// TwinCAT 3 PLC project test
// ProgramVersion: 3.1.4020.5
// libraries:
//   L2Si Vacuum Library, * (SLAC)
//   LCLS General, * (SLAC)
//   PMPS, * (SLAC - LCLS)
//   Tc2_Standard, * (Beckhoff Automation GmbH)
//   Tc2_System, * (Beckhoff Automation GmbH)
//   Tc2_Utilities, * (Beckhoff Automation GmbH)
//   Tc3_Module, * (Beckhoff Automation GmbH)
// project tree:
//   DUTs/ E_STATES.TcTLEO
//   GVLs/ GVL_Devices.TcGVL, GVL_PMPS.TcGVL
//   / PlcTask.TcTTO
//   POUs/ FB_ValveBase.TcPOU, FB_VGC.TcPOU, FB_VGC_FFO.TcPOU, FB_VRC_NO.TcPOU, MAIN.TcPOU, PRG_VLS.TcPOU
// real-time tasks:
//   TASK PlcTask: cycle T#10ms, priority 20, ADS port 350
//   TASK SimTask: cycle T#10ms, priority 1, ADS port 351
//   TASK VacTask: cycle T#10ms, priority 2, ADS port 352
// I/O:
//   DEVICE Device 1 (EtherCAT) (disabled), AmsNetId 172.21.148.60.2.1
//     Term 1 (EK1100) [EK1100 EtherCAT Coupler (2A E-Bus)]
//       Term 2 (EL3174-0002) [EL3174-0002 4Ch. Ana. Input +/-10V, +/-20mA 16 Bit, Isolated Channels]
//       Term 3 (EL3174-0002) [EL3174-0002 4Ch. Ana. Input +/-10V, +/-20mA 16 Bit, Isolated Channels]
//       Term 4 (EL2624) [EL2624 4Ch. Relay Output, NO (125V AC / 30V DC)]
//       Term 6 (EL1004) [EL1004 4Ch. Dig. Input 24V, 3ms]
//       Term 5 (EL1004) [EL1004 4Ch. Dig. Input 24V, 3ms]
//       Term 7 (EL2004) [EL2004 4Ch. Dig. Output 24V, 0.5A]
//       Term 8 (EL3064) [EL3064 4Ch. Ana. Input 0-10V]
//       Term 9 (EL2794) [EL2794 4Ch. Dig. Output 24V AC/DC, 2A, short-circuit-proof]
//       Term 10 (EL1004) [EL1004 4Ch. Dig. Input 24V, 3ms]
//       Term 11 (EL1124) [EL1124 4Ch. Dig. Input 5V, 10µs, Sensor Power]
//       Term 12 (EL1124) [EL1124 4Ch. Dig. Input 5V, 10µs, Sensor Power]
//       Term 13 (EL3064) [EL3064 4Ch. Ana. Input 0-10V]
// variable links:
//   SIM/SIM Instance <-> test/test Instance
//     PlcTaskSim Inputs/GVL_SimDevices.S_FEE_GCC_03.i_xHvOn <-> PlcTask Outputs/GVL_Devices.FEE_GCC_03.q_xHV_DIS
//     PlcTaskSim Inputs/GVL_SimDevices.S_FEE_GCC_04.i_xHvOn <-> PlcTask Outputs/GVL_Devices.FEE_GCC_04.q_xHV_DIS
//     PlcTaskSim Inputs/GVL_SimDevices.S_FEE_KMONO_GCC_01.i_xHvOn <-> PlcTask Outputs/GVL_Devices.FEE_KMONO_GCC_01.q_xHV_DIS
//     PlcTaskSim Inputs/GVL_SimDevices.S_FEE_KMONO_PIP_01.xOn <-> PlcTask Outputs/GVL_Devices.FEE_KMONO_PIP_01.q_xHVEna_DO
//     PlcTaskSim Inputs/GVL_SimDevices.S_FEE_M1L_PIP_01.xOn <-> PlcTask Outputs/GVL_Devices.FEE_M1L_PIP_01.q_xHVEna_DO
//     PlcTaskSim Inputs/GVL_SimDevices.S_FEE_MIL_GCC_02.i_xHvOn <-> PlcTask Outputs/GVL_Devices.FEE_M1L_GCC_01.q_xHV_DIS
//     PlcTaskSim Inputs/GVL_SimDevices.S_FEE_PIP_02.xOn <-> PlcTask Outputs/GVL_Devices.FEE_PIP_02.q_xHVEna_DO
//     PlcTaskSim Inputs/GVL_SimDevices.S_FEE_PIP_03.xOn <-> PlcTask Outputs/GVL_Devices.FEE_PIP_03.q_xHVEna_DO
//     PlcTaskSim Inputs/GVL_SimDevices.S_FEE_VGC_02.i_xSol <-> PlcTask Outputs/GVL_Devices.FEE_VGC_02.q_xOPN_DO
//     PlcTaskSim Inputs/GVL_SimDevices.S_FEE_VGC_03.i_xSol <-> PlcTask Outputs/GVL_Devices.FEE_VGC_03.q_xOPN_DO
//     PlcTaskSim Inputs/GVL_SimDevices.S_FEE_VGC_04.i_xSol <-> PlcTask Outputs/GVL_Devices.FEE_VGC_04.q_xOPN_DO
//     PlcTaskSim Inputs/GVL_SimDevices.VGC_1.i_xSol <-> PlcTask Outputs/PRG_VLS.VGC_1.q_xOPN_DO
//     PlcTaskSim Inputs/GVL_SimDevices.VGC_W.i_xSol <-> PlcTask Outputs/PRG_VLS.VGC_W.q_xCLS_DO
//     PlcTaskSim Outputs/GVL_SimDevices.S_FEE_GCC_03.q_DisActive <-> PlcTask Inputs/GVL_Devices.FEE_GCC_03.i_xDisc_Active
//     PlcTaskSim Outputs/GVL_SimDevices.S_FEE_GCC_04.q_DisActive <-> PlcTask Inputs/GVL_Devices.FEE_GCC_04.i_xDisc_Active
//     PlcTaskSim Outputs/GVL_SimDevices.S_FEE_GCC_03.q_iRawPress <-> PlcTask Inputs/GVL_Devices.FEE_GCC_03.i_iPRESS_R
//     PlcTaskSim Outputs/GVL_SimDevices.S_FEE_GCC_04.q_iRawPress <-> PlcTask Inputs/GVL_Devices.FEE_GCC_04.i_iPRESS_R
//     PlcTaskSim Outputs/GVL_SimDevices.S_FEE_GCC_03.q_iRawPress <-> PlcTask Inputs/PRG_VLS.DS_GCC.i_iPRESS_R
//     PlcTaskSim Outputs/GVL_SimDevices.S_FEE_GCC_03.q_xHVOn <-> PlcTask Inputs/GVL_Devices.FEE_GCC_03.i_xHV_ON
//     PlcTaskSim Outputs/GVL_SimDevices.S_FEE_GCC_04.q_xHVOn <-> PlcTask Inputs/GVL_Devices.FEE_GCC_04.i_xHV_ON
//     PlcTaskSim Outputs/GVL_SimDevices.S_FEE_GPI_03.q_iRawPress <-> PlcTask Inputs/GVL_Devices.FEE_GPI_03.i_iPRESS_R
//     PlcTaskSim Outputs/GVL_SimDevices.S_FEE_GPI_04.q_iRawPress <-> PlcTask Inputs/GVL_Devices.FEE_GPI_04.i_iPRESS_R
//     PlcTaskSim Outputs/GVL_SimDevices.S_FEE_GPI_03.q_iRawPress <-> PlcTask Inputs/PRG_VLS.DS_GPI.i_iPRESS_R
//     PlcTaskSim Outputs/GVL_SimDevices.S_FEE_KMONO_GCC_01.q_DisActive <-> PlcTask Inputs/GVL_Devices.FEE_KMONO_GCC_01.i_xDisc_Active
//     PlcTaskSim Outputs/GVL_SimDevices.S_FEE_KMONO_GCC_01.q_iRawPress <-> PlcTask Inputs/GVL_Devices.FEE_KMONO_GCC_01.i_iPRESS_R
//     PlcTaskSim Outputs/GVL_SimDevices.S_FEE_KMONO_GCC_01.q_iRawPress <-> PlcTask Inputs/PRG_VLS.US_GCC.i_iPRESS_R
//     PlcTaskSim Outputs/GVL_SimDevices.S_FEE_KMONO_GCC_01.q_xHVOn <-> PlcTask Inputs/GVL_Devices.FEE_KMONO_GCC_01.i_xHV_ON
//     PlcTaskSim Outputs/GVL_SimDevices.S_FEE_KMONO_GPI_01.q_iRawPress <-> PlcTask Inputs/GVL_Devices.FEE_KMONO_GPI_01.i_iPRESS_R
//     PlcTaskSim Outputs/GVL_SimDevices.S_FEE_KMONO_GPI_01.q_iRawPress <-> PlcTask Inputs/PRG_VLS.US_GPI.i_iPRESS_R
//     PlcTaskSim Outputs/GVL_SimDevices.S_FEE_M1L_GPI_02.q_iRawPress <-> PlcTask Inputs/GVL_Devices.FEE_M1L_GPI_01.i_iPRESS_R
//     PlcTaskSim Outputs/GVL_SimDevices.S_FEE_MIL_GCC_02.q_DisActive <-> PlcTask Inputs/GVL_Devices.FEE_M1L_GCC_01.i_xDisc_Active
//     PlcTaskSim Outputs/GVL_SimDevices.S_FEE_MIL_GCC_02.q_iRawPress <-> PlcTask Inputs/GVL_Devices.FEE_M1L_GCC_01.i_iPRESS_R
//     PlcTaskSim Outputs/GVL_SimDevices.S_FEE_MIL_GCC_02.q_xHVOn <-> PlcTask Inputs/GVL_Devices.FEE_M1L_GCC_01.i_xHV_ON
//     PlcTaskSim Outputs/GVL_SimDevices.S_FEE_VGC_02.q_xClsLS <-> PlcTask Inputs/GVL_Devices.FEE_VGC_02.i_xClsLS
//     PlcTaskSim Outputs/GVL_SimDevices.S_FEE_VGC_03.q_xClsLS <-> PlcTask Inputs/GVL_Devices.FEE_VGC_03.i_xClsLS
//     PlcTaskSim Outputs/GVL_SimDevices.S_FEE_VGC_04.q_xClsLS <-> PlcTask Inputs/GVL_Devices.FEE_VGC_04.i_xClsLS
//     PlcTaskSim Outputs/GVL_SimDevices.S_FEE_VGC_02.q_xOpnLS <-> PlcTask Inputs/GVL_Devices.FEE_VGC_02.i_xOpnLS
//     PlcTaskSim Outputs/GVL_SimDevices.S_FEE_VGC_03.q_xOpnLS <-> PlcTask Inputs/GVL_Devices.FEE_VGC_03.i_xOpnLS
//     PlcTaskSim Outputs/GVL_SimDevices.S_FEE_VGC_04.q_xOpnLS <-> PlcTask Inputs/GVL_Devices.FEE_VGC_04.i_xOpnLS
//     PlcTaskSim Outputs/GVL_SimDevices.VGC_1.q_xClsLS <-> PlcTask Inputs/PRG_VLS.VGC_1.i_xClsLS
//     PlcTaskSim Outputs/GVL_SimDevices.VGC_1.q_xOpnLS <-> PlcTask Inputs/PRG_VLS.VGC_1.i_xOpnLS
//     PlcTaskSim Outputs/GVL_SimDevices.VGC_W.q_xClsLS <-> PlcTask Inputs/PRG_VLS.VGC_W.i_xClsLS
//     PlcTaskSim Outputs/GVL_SimDevices.VGC_W.q_xOpnLS <-> PlcTask Inputs/PRG_VLS.VGC_W.i_xOpnLS

CONFIGURATION test
    RESOURCE PLC ON TwinCAT3
        TASK PlcTask(INTERVAL := T#10ms, PRIORITY := 2);
        PROGRAM MAIN WITH PlcTask : MAIN;
    END_RESOURCE
END_CONFIGURATION

// ---- DUTs/E_STATES.TcTLEO
{attribute 'qualified_only'}
{attribute 'strict'}
TYPE E_STATES :
(
	INIT := 0, // INIT 
	NOT_SAFE ,// NOT OK to move in the same state
	READY, // Safe to Move STATE
	OVERRIDE,
	SETUP
	
);
END_TYPE

// ---- GVLs/GVL_Devices.TcGVL
VAR_GLOBAL
	
	

/////////////////////
	{attribute 'pytmc' := '
    pv: FEE:VGC:02
	'}
	FEE_VGC_02: FB_VGC;
	{attribute 'pytmc' := '
    pv: FEE:KMONO:GPI:01
	'}
	FEE_KMONO_GPI_01: FB_MKS275;
	{attribute 'pytmc' := '
    pv: FEE:KMONO:GCC:01
	'}
	FEE_KMONO_GCC_01: FB_MKS500;
	{attribute 'pytmc' := '
    pv: FEE:KMONO:PIP:01
	'}
	FEE_KMONO_PIP_01: FB_PIP_Gamma;
	{attribute 'pytmc' := '
    pv: FEE:PIP:02
	'}
	FEE_PIP_02: FB_PIP_Gamma;
	{attribute 'pytmc' := '
    pv: FEE:GPI:03
	'}
	FEE_GPI_03: FB_MKS275;
	{attribute 'pytmc' := '
    pv: FEE:GCC:03
	'}
	FEE_GCC_03: FB_MKS500;
	{attribute 'pytmc' := '
    pv: FEE:VGC:03
	'}
	FEE_VGC_03: FB_VGC_FFO;
	{attribute 'pytmc' := '
    pv: FEE:M1L:GPI:01
	'}
	FEE_M1L_GPI_01: FB_MKS275;
	{attribute 'pytmc' := '
    pv: FEE:M1L:GCC:03
	'}
	FEE_M1L_GCC_01: FB_MKS500;
	{attribute 'pytmc' := '
    pv: FEE:M1L:PIP:01
	'}
	FEE_M1L_PIP_01: FB_PIP_Gamma;
	{attribute 'pytmc' := '
    pv: FEE:PIP:03
	'}
	FEE_PIP_03: FB_PIP_Gamma;
	{attribute 'pytmc' := '
    pv: FEE:GPI:04
	'}
	FEE_GPI_04: FB_MKS275;
	{attribute 'pytmc' := '
    pv: FEE:GCC:04
	'}
	FEE_GCC_04: FB_MKS500;
	{attribute 'pytmc' := '
    pv: FEE:VGC:04
	'}
	FEE_VGC_04: FB_VGC_FFO;
	
END_VAR

// ---- GVLs/GVL_PMPS.TcGVL

VAR_GLOBAL
	
{attribute 'pytmc' := '
    pv: PLC:TST:FF1
    '}
    {attribute 'TcLinkTo' := '.q_xFastFaultOut:=TIIB[PMPS_FFO]^Channel 1^Output'}
    g_FastFaultOutput1  :   FB_HardwareFFOutput;
	
	{attribute 'pytmc' := '
    pv: PLC:TST:FF2
    '}
    {attribute 'TcLinkTo' := '.q_xFastFaultOut:=TIIB[PMPS_FFO]^Channel 2^Output'}
    g_FastFaultOutput2  :   FB_HardwareFFOutput;
END_VAR

// ---- POUs/MAIN.TcPOU
PROGRAM MAIN
VAR
	
	

END_VAR

PRG_VLS();

//valves
FEE_VGC_02(
	i_stUSG:= FEE_KMONO_GCC_01.IG, 
	i_stDSG:= FEE_KMONO_GCC_01.IG , 
	i_xDis_DPIlk:= FALSE, 
	i_xEPS_OPN_OK:= , 
	i_xEPS_CLS_OK:= ,
	i_xPMPS_OK:= , 
	i_xExt_OK:= TRUE, 
	i_xOverrideMode:= , 
	i_xReset:= , 
	iq_stValve=>);

FEE_VGC_03(
	i_stUSG:=FEE_KMONO_GCC_01.IG, 
	i_stDSG:= FEE_M1L_GCC_01.IG , 
	i_xDis_DPIlk:= FALSE, 
	i_xEPS_OPN_OK:= TRUE, 
	i_xEPS_CLS_OK:= TRUE,
	i_xPMPS_OK:= TRUE, 
	i_xExt_OK:= TRUE, 
	i_xOverrideMode:= , 
	i_xReset:= , 
	iq_stValve=> , 
	xMPS_OK=> , 
	io_fbFFHWO:= g_FastFaultOutput1 );

FEE_VGC_04(
	i_stUSG:= FEE_GCC_03.IG, 
	i_stDSG:= FEE_GCC_03.IG , 
	i_xDis_DPIlk:= FALSE, 
	i_xEPS_OPN_OK:= TRUE, 
	i_xEPS_CLS_OK:= TRUE,
	i_xPMPS_OK:= TRUE, 
	i_xExt_OK:= TRUE, 
	i_xOverrideMode:= , 
	i_xReset:= , 
	iq_stValve=> , 
	xMPS_OK=> , 
	io_fbFFHWO:= g_FastFaultOutput2 );	
	
// gauges and pip
FEE_KMONO_GPI_01(PG=>);
FEE_KMONO_GCC_01(PG:=FEE_KMONO_GPI_01.PG);
FEE_KMONO_PIP_01(i_stGauge:= FEE_KMONO_GCC_01.IG);

FEE_GPI_03(PG=>);
FEE_GCC_03(PG:=FEE_KMONO_GPI_01.PG);

FEE_PIP_02(i_stGauge:= FEE_GCC_03.IG);

FEE_M1L_GPI_01(PG=>);
FEE_M1L_GCC_01(PG:=FEE_M1L_GPI_01.PG);
FEE_M1L_PIP_01(i_stGauge:= FEE_M1L_GCC_01.IG);

FEE_GPI_04(PG=>);
FEE_GCC_04(PG:=FEE_GPI_04.PG);
FEE_PIP_03(i_stGauge:= FEE_GCC_04.IG);



/// fast fault

g_FastFaultOutput1.EvaluateOutput(i_xVeto:=PMPS_GVL.stCurrentBeamParameters.aStoppers[PMPS.L_Stopper.ST1]);
g_FastFaultOutput2.EvaluateOutput(i_xVeto:=PMPS_GVL.stCurrentBeamParameters.aStoppers[PMPS.L_Stopper.ST1]);

END_PROGRAM

// ---- POUs/PRG_VLS.TcPOU
PROGRAM PRG_VLS
VAR
	xFirstPass	:	BOOL;
	fbFSInit		:	R_TRIG;
	
	state:E_STATES;
	

	bOverride:BOOL;
	bSetup:BOOL;
	
	
	//GVL_Devices
	VGC_1	:FB_VGC;
	VGC_W	:FB_VRC_NO; // Is the Window valve NO 

	US_GPI: FB_MKS275;
	US_GCC: FB_MKS422;

	DS_GPI: FB_MKS275;
	DS_GCC: FB_MKS422;
END_VAR

fbFSInit( CLK := TRUE, Q => xFirstPass);
(* On first PLC pass, put valve into init state*)
IF xFirstPass THEN
	state:= E_STATES.INIT;
	bOverride := FALSE;
	bSetup := FALSE;
END_IF


//STATE ACTIONS
CASE state OF

 E_STATES.INIT: 
		VGC_1.M_Set_OPN_SW(FALSE); //Isolation Valve closed
		VGC_W.M_Set_CLS_SW(FALSE); // Window valve OPEN
		VGC_1.i_xOverrideMode := VGC_W.i_xOverrideMode := FALSE;
		//Transition
		if (VGC_1.M_IsClosed() AND VGC_W.M_IsOpen()) THEN
			state:= E_STATES.NOT_SAFE;
		END_IF
		
E_STATES.NOT_SAFE: // System is not allowed to actuate, i.e all interlocks are in effect
 	VGC_1.i_xExt_OK := VGC_1.i_xEPS_OPN_OK := VGC_1.i_xEPS_CLS_OK:= FALSE; 
	VGC_W.i_xExtILK_OK:= FALSE; 
	VGC_1.i_xOverrideMode := VGC_W.i_xOverrideMode := FALSE;

	//Transition
	if (US_GCC.IG.xAT_VAC AND DS_GCC.IG.xAT_VAC) THEN state:= E_STATES.READY; END_IF
	
	
 E_STATES.READY: // OK to MOVE
 	// Release the external interlock so the differential pressure inlk is in effect
 	VGC_1.i_xExt_OK:= VGC_1.i_xEPS_OPN_OK := VGC_1.i_xEPS_CLS_OK:= TRUE; 
	//permission to insert window valve only when US vacuum is good??
	VGC_W.i_xExtILK_OK:= US_GCC.IG.xPRESS_OK AND  US_GCC.IG.xAT_VAC; // OR should it be a pressure setpoint
	//Insertion of window valve is followed by automatic openeing of isolation valve.
	// Valves  alternate positions.
	If (VGC_W.M_IsClosed()) THEN  VGC_1.M_Set_OPN_SW(TRUE);
	ELSIF (VGC_W.M_IsOpen()) THEN VGC_1.M_Set_OPN_SW(FALSE);
	END_IF
	
 
 E_STATES.OVERRIDE: 
	// Override Mode is enabled for all valves
 	VGC_1.i_xOverrideMode :=VGC_W.i_xOverrideMode := TRUE;
	// Exit of Override mode always goes back to init
 	IF NOT(bOverride) THEN state:= E_STATES.INIT; END_IF
	
	
 E_STATES.SETUP: 
	// Window valve remains retracted
 	VGC_W.i_xExtILK_OK := FALSE; 
	// Isolation valves operates like standard gate valves 
	VGC_1.i_xExt_OK := TRUE;
	// exit to init just to be safe?
	IF NOT(bSetup) THEN state:= E_STATES.INIT; END_IF
END_CASE





// STATE TRANSITIONS
// the system can go to setup state from any other state except override
IF (bSetup) AND (state<>E_STATES.OVERRIDE) THEN state:= E_STATES.SETUP; 
// the system can go to override state from any other state except setup
ELSIF (bOverride) AND (state<>E_STATES.SETUP) THEN state:= E_STATES.OVERRIDE;
//Loss of at vac signal makes the system go to init/not safe to move state
ELSIF (NOT US_GCC.IG.xAT_VAC ) OR (NOT DS_GCC.IG.xAT_VAC) THEN state:= E_STATES.INIT;
END_IF 





// Instantiate function blocks
US_GPI(PG=>);
US_GCC(PG:=US_GPI.PG);
DS_GPI(PG=>);
DS_GCC(PG:=US_GPI.PG);

VGC_1(
	i_stUSG:= US_GCC.IG, 
	i_stDSG:= DS_GCC.IG , 
	i_xDis_DPIlk:= FALSE, 
	i_xEPS_OPN_OK:= , 
	i_xEPS_CLS_OK:= ,
	i_xPMPS_OK:= , 
	i_xExt_OK:= , 
	i_xOverrideMode:= , 
	i_xReset:= , 
	iq_stValve=>);

VGC_W(i_xExtILK_OK:= , 
	i_xOverrideMode:= ,
    iq_stValve=> );

END_PROGRAM

// ---- POUs/FB_VGC.TcPOU
(* This function block implements basic functionality for Isolation Gate Valves*)
(* This function block interlock is as follows:
1. The valve can be opened when the difference between the pressures on both sides is
less than the maximum differential pressure.
2. This rule persists until the pressures on both sides are lower than the vacuum-setpoint.
3. Once at-vac, the valve will close if the pressure on either side rises above the setpoint.*)
(*This function block also implements PMPS and EPS interlocks, as well as Fast MPS trigger*)
FUNCTION_BLOCK FB_VGC Extends FB_ValveBase
VAR_IN_OUT
END_VAR
VAR_INPUT
	(*Upstream Gauge, usually ion gauge*)
	i_stUSG	:	ST_VG;
	(*Downstream Gauge, usually ion gauge*)
	i_stDSG	:	ST_VG;
	{attribute 'pytmc' := '
    pv: Dis_DPIlk
	'}
	i_xDis_DPIlk : BOOL := FALSE;  (* Set to true when calling the function to disable the differential pressure interlock *)
	{attribute 'pytmc' := '
    pv: EPS_OPN_OK
	'}
	i_xEPS_OPN_OK:	BOOL	:= TRUE; (*External EPS interlock, Set to TRUE when no EPS interlock is required, otherwise set to correct interlock signal*)
	{attribute 'pytmc' := '
    pv: EPS_CLS_OK
	'}
	i_xEPS_CLS_OK:	BOOL	:= TRUE; (*External EPS interlock, Set to TRUE when no EPS interlock is required, otherwise set to correct interlock signal*)
	
	{attribute 'pytmc' := '
    pv: MPS_OK
	'}
	i_xPMPS_OK:	BOOL	; (*External MPS interlock, Set to TRUE when no PMPS interlock is required*)
	i_xExt_OK: BOOL; (*Other External Interlock, Set to True when no external interlock is required. If this Valve is neigboring a Fast Shutter this should be linked to the fast shutter xVAC_FAULT_OK*)
	i_xOverrideMode : BOOL; (*To be linked to global override bit. This Overrides Vacuum logic only, EPS, MPS and PMPS are still enforces*)
	// Reset fault
	{attribute 'pytmc' := '
    pv: FF_Reset
	'}
    i_xReset: BOOL;
END_VAR
VAR_OUTPUT
	{attribute 'pytmc' := '
    pv:
	'}
	iq_stValve : ST_VGC; (* All valve data and states will be in this struct*)
	
END_VAR

VAR
	{attribute 'instance-path'}
	{attribute 'noinit'}
	sPath: STRING;
	rDiffPressAllowed	:	REAL := 22.5; // Torr, Default value comes from Vat Valve Manual
	rDiffPress : REAL;
	set : BOOL;
    reset: BOOL;
	  
	xFirstPass	:	BOOL;
	fbFSInit		:	R_TRIG;
	
	tonDelOK : TON;
	rtOK	:	R_TRIG;
	tonOvrd	:	TON;
	rtOpen	:	R_TRIG;
	ftClose: F_TRIG;
	
	tDelOK	:	TIME := T#60S;
	tOvrd	:	TIME := T#10s;
	ePrevState : E_VGC;
	
	(* Timeouts*)
	tTimeOutDuration: TIME:= T#10S;
	tOPNtimeout: TON;
	tCLStimeout:TON;
	
	
	
	(*IO*)
	i_xOpnLS	AT%I*: BOOL;
	i_xClsLS	AT%I*: BOOL;
	q_xOPN_DO	AT%Q*: BOOL;
    
  
END_VAR

(* Vacuum gate valve
A. Wallace
16-10-29

A gate valve isolates vacuum volumes. Ideally it can be opened when a system is vented
to allow for faster pumping, and will close when high vacuum is lost.

The following behavior is good for valves in something like a gas attenuator.
This function block does the following:
1. The valve can be opened when the difference between the pressures on both sides is
less than the maximum differential pressure.
2. This rule persists until the pressures on both sides are lower than the vacuum-setpoint.
3. Once at-vac, the valve will close if the pressure on either side rises above the setpoint.

Alternatively, the differential pressure interlock can be disabled so the valve may only be opened
if the pressure on both sides is lower than the at-vacuum-setpoint. You want this behavior if 
the valve is to be used in a UHV section.

Hysteresis is employed to ensure a smooth transition from vented/pumping down, to at-vac.

Finally, an override system is built in so you can bypass all the interlocking logic and 
get back online.
*)
(* 10/1/2018 Margaret Ghaly included EPS, PMPS Checkes and MPS trigger signals*)

ACT_Init();
(*IO Mapping*)
ACT_IO();
A_Override();
A_PositionCheck();
ACT_ResetAlarms();
A_EPS();
// Main logic the very last call right before IO
ACT_Main();
(*IO Mapping*)
ACT_IO();
A_Logger();

ACTION A_EPS:
ftClose(CLK:= iq_stValve.pv_xOPN_SW);
rtOpen(CLK:= iq_stValve.pv_xOPN_SW);


(* If Epics Command to close the Valve, check if PMPS and EPS are ok, otherwise Keep command set to open valve *)
// Check a falling edge on the open switch, which means that the valve is commanded to close
IF (ftClose.Q) THEN
	// check that the valve is allowed to close, and that it was already in the open position otherwise, he command is to be ingonred and reset
	IF NOT(i_xEPS_CLS_OK) AND (iq_stValve.q_xOPN_DO) THEN iq_stValve.pv_xOPN_SW := TRUE; END_IF;
END_IF

// if switch pv has been switched to open
IF (rtOpen.Q) THEN 
	// if the EPS interlock the valve from openening, the switch pv is reset to false i.e ignoring the action
	IF NOT (i_xEPS_OPN_OK) THEN  iq_stValve.pv_xOPN_SW := FALSE; END_IF
END_IF
END_ACTION

ACTION A_Logger:
// Log valve timeouts
tErrorPresent(CLK:=iq_stValve.bErrorPresent);
IF tErrorPresent.Q THEN fbLogger(sMsg:=iq_stValve.sErrorMessage, eSevr:=TcEventSeverity.Warning); END_IF

// Log valve open
tAction(CLK:= iq_stValve.q_xOPN_DO);
IF tAction.Q THEN fbLogger(sMsg:='Valve commanded open', eSevr:=TcEventSeverity.Info); END_IF

// Log override mode enabled
tOverrideActivated(CLK:= (tonOvrd.Q AND i_xOverrideMode));
IF tOverrideActivated.Q THEN fbLogger(sMsg:='Valve override mode activated', eSevr:=TcEventSeverity.Warning); END_IF
END_ACTION

ACTION A_Override:
(* Override logic *)
(* Goal: give ability to override, but do so in a way that people won't forget it.
Solution: Override only after ten seconds of override, protect against blips,
when the valve permission goes true for more than ten seconds consistently, remove override
*)

tonDelOK(IN:=iq_stValve.xOPN_OK, PT:=tDelOK);
rtOK(CLK:=tonDelOK.Q);
IF rtOK.Q AND iq_stValve.pv_xOvrdOpn THEN 
	if (iq_stValve.eState = OPEN) AND (i_xOverrideMode) AND (iq_stValve.pv_xOvrdOpn) THEN iq_stValve.pv_xOPN_SW := TRUE; END_IF //for seamless transition   
   	iq_stValve.pv_xOvrdOpn :=FALSE; // reset the overrride open bit
	//Log
    fbLogger(sMsg:='Override expired', eSevr:=TcEventSeverity.Warning);
    
END_IF

//Override timer
tonOvrd(IN:=iq_stValve.pv_xOvrdOpn, PT:=tOvrd);
END_ACTION

ACTION A_PositionCheck:


///Check valve position
IF iq_stValve.i_xClsLS AND  iq_stValve.i_xOpnLS THEN
	iq_stValve.eState:=INVALID;
ELSIF NOT iq_stValve.i_xClsLS AND iq_stValve.i_xOpnLS AND iq_stValve.q_xOPN_DO THEN 
	iq_stValve.eState:=OPEN;
ELSIF iq_stValve.i_xClsLS AND NOT iq_stValve.i_xOpnLS AND NOT iq_stValve.q_xOPN_DO THEN 
	iq_stValve.eState:=CLOSED;
ELSIF NOT iq_stValve.i_xClsLS AND NOT iq_stValve.i_xOpnLS THEN 
	iq_stValve.eState:=MOVING;
ELSE
	iq_stValve.eState:=INVALID;
END_IF


///Check valve moving postion timout
IF NOT iq_stValve.i_xClsLS AND tCLStimeout.Q THEN 
	iq_stValve.bErrorPresent := TRUE;
	iq_stValve.sErrorMessage := ' Close Timeout';
ELSIF NOT iq_stValve.i_xOpnLS AND tOPNtimeout.Q THEN 
	iq_stValve.bErrorPresent := TRUE; 
	iq_stValve.sErrorMessage := ' Open Timeout';
END_IF
IF (iq_stValve.eState=INVALID) THEN
	iq_stValve.bErrorPresent := TRUE; 
	iq_stValve.sErrorMessage := CONCAT(sPath,' Invalid Valve Position');
END_IF


(*Timers*)
tOPNtimeout(IN:= iq_stValve.q_xOPN_DO, PT := tTimeOutDuration );
tCLStimeout(IN:= NOT iq_stValve.q_xOPN_DO, PT := tTimeOutDuration);
END_ACTION

ACTION ACT_Init:
fbFSInit( CLK := TRUE, Q => xFirstPass);
(* On first PLC pass, put valve into vented state, which implies a closed valve *)
IF xFirstPass THEN
	iq_stValve.eVGC_State := Vented;
	iq_stValve.pv_xOPN_SW := FALSE;
END_IF
END_ACTION

ACTION ACT_IO:
(*inputs*)
iq_stValve.i_xOpnLS := 	i_xOpnLS;
iq_stValve.i_xClsLS:=	i_xClsLS;
iq_stValve.xEXT_OK := i_xEXT_OK;
iq_stValve.xOverrideMode := i_xOverrideMode;
(*outputs*)
q_xOPN_DO:= iq_stValve.q_xOPN_DO;
END_ACTION

ACTION ACT_Main:

// Update hysteresis
///////////////////////////////////////////////////
IF iq_stValve.rAT_VAC_SP_LAST <> iq_stValve.rAT_VAC_SP OR xFirstPass THEN
	iq_stValve.rAT_VAC_SP_LAST := iq_stValve.rAT_VAC_SP;
	iq_stValve.rAT_VAC_HYS := iq_stValve.rHYST_PERC * iq_stValve.rAT_VAC_SP;
END_IF

iq_stValve.rAT_VAC_HYS := LIMIT(0, iq_stValve.rAT_VAC_HYS, iq_stValve.rAT_VAC_SP);
IF iq_stValve.rAT_VAC_SP <> 0 THEN
	IF iq_stValve.rHYST_PERC <> (iq_stValve.rAT_VAC_HYS / iq_stValve.rAT_VAC_SP) THEN
		iq_stValve.rHYST_PERC := LIMIT(0, (iq_stValve.rAT_VAC_HYS / iq_stValve.rAT_VAC_SP) ,1);
	END_IF
END_IF
// Valve at vacuum check
///////////////////////////////////////////////////
	set := i_stUSG.rPRESS < iq_stValve.rAT_VAC_HYS AND i_stDSG.rPRESS < iq_stValve.rAT_VAC_HYS AND i_stUSG.xPRESS_OK AND i_stDSG.xPRESS_OK;
 	iq_stValve.xAT_VAC S= set;
	reset := i_stUSG.rPRESS > iq_stValve.rAT_VAC_SP OR i_stDSG.rPRESS > iq_stValve.rAT_VAC_SP OR NOT i_stUSG.xPRESS_OK OR NOT i_stDSG.xPRESS_OK;
	iq_stValve.xAT_VAC R= reset;
	
// Differential pressure check
///////////////////////////////////////////////////
	(* Calc the differential pressure across the valve *)
	rDiffPress := ABS(i_stUSG.rPRESS - i_stDSG.rPRESS);
	
	(* As long as the differential pressure is less than 30mbar, the valve is allowed to open *)
	IF rDiffPress <= rDiffPressAllowed AND i_stUSG.xPRESS_OK AND i_stDSG.xPRESS_OK THEN
		iq_stValve.xDP_OK := TRUE;
	ELSE
		iq_stValve.xDP_OK	:= FALSE;
		(* If the differential pressure is exceeded, even when the valve is open,
		the state is unexpected and triggers a fault, because it suggests that something
		is wrong with the valve, or gauges or mapping or there is a major leak on one side.*)
		iq_stValve.eVGC_State := ERR_DiffPress;
        iq_stValve.xERR_DifPres := TRUE;
	END_IF

// Valve state
///////////////////////////////////////////////////
CASE iq_stValve.eVGC_State OF
	Vented: (* The Vented state is used during pump down *)
        //Log new state
        IF ePrevState <> iq_stValve.eVGC_State THEN
            fbLogger(sMsg:='Vented', eSevr:=TcEventSeverity.Info);
            ePrevState := iq_stValve.eVGC_State;
		END_IF
        
		(* Assuming the pump down went well, we are now at vacuum on both sides,
		so we move to the vacuum state, otherwise remain in the vented state *)
		IF iq_stValve.xAT_VAC AND (NOT (iq_stValve.xERR_DifPres)) AND NOT (NOT (iq_stValve.xERR_SP)) and NOT (NOT (iq_stValve.xERR_ExtFault))THEN
		    iq_stValve.eVGC_State := AtVacuum;
		ELSE
		    iq_stValve.eVGC_State := Vented;
		END_IF
	
	AtVacuum:
        //Log new state
        IF ePrevState <> iq_stValve.eVGC_State THEN
            fbLogger(sMsg:='Vacuum setpoint satisfied', eSevr:=TcEventSeverity.Info);
            ePrevState := iq_stValve.eVGC_State;
		END_IF
        
		IF iq_stValve.xAT_VAC THEN
		(* If both pressure setpoints are made,
		then enable the differential pressure interlock, regardless of the valve state
		assuming we're using some kind of ion gauge where a pressure setpoint cannot be higher than 1E-4 T *)
		iq_stValve.eVGC_State := AtVacuum;
				
		ELSE
		
			(* If the valve is open (or in an unknown state) and either gauge is not at it's vacuum setpoint,
			we have a loss of vacuum error *)
			IF (iq_stValve.i_xOpnLS OR (NOT iq_stValve.i_xOpnLS AND NOT iq_stValve.i_xClsLS)) THEN
				iq_stValve.eVGC_State := ERR_LostVac;
				iq_stValve.xERR_SP := TRUE; //TAW changed this to the ERR_SP bool because I think that's what it was intended to be?
		
			(* Alternatively, if the valve is already closed and we lose pressure on one side,
			it was probably intentional venting, so we calmly move back to venting mode, and
			disable the differential pressure interlock *) //?? 
			ELSIF iq_stValve.i_xClsLS THEN
				iq_stValve.eVGC_State := Vented;
			END_IF
		
		END_IF
	
	ERR_DiffPress:
        //Log new state
        IF ePrevState <> iq_stValve.eVGC_State THEN
            fbLogger(sMsg:='Potential accidental vent.', eSevr:=TcEventSeverity.Critical);
            ePrevState := iq_stValve.eVGC_State;
		END_IF
        
		IF NOT (iq_stValve.xERR_DifPres) THEN
			iq_stValve.eVGC_State := Vented;
		END_IF
		
	
	ERR_LostVac:
        //Log new state
        IF ePrevState <> iq_stValve.eVGC_State THEN
            fbLogger(sMsg:='Unexpected loss of vacuum while valve was open.', eSevr:=TcEventSeverity.Critical);
            ePrevState := iq_stValve.eVGC_State;
		END_IF
		IF NOT (iq_stValve.xERR_SP) THEN
			iq_stValve.eVGC_State := Vented;
		END_IF
		
	ERR_ExtFault:
        //Log new state
        IF ePrevState <> iq_stValve.eVGC_State THEN
            fbLogger(sMsg:='Lost external interlock while valve was open.', eSevr:=TcEventSeverity.Critical);
            ePrevState := iq_stValve.eVGC_State;
		END_IF
		IF NOT (iq_stValve.xERR_ExtFault) AND (NOT i_xExt_OK) THEN
			iq_stValve.eVGC_State := Vented;
		END_IF
END_CASE

IF (NOT i_xExt_OK) THEN
	iq_stValve.eVGC_State := ERR_ExtFault;
	iq_stValve.xERR_ExtFault := TRUE;
END_IF

// Interlock evaluation - with bypass for DP ILK bypass
///////////////////////////////////////////////
IF i_xDis_DPIlk THEN
	iq_stValve.xOPN_OK := iq_stValve.xEXT_OK; // AND iq_stValve.xDP_OK ;
ELSE
	iq_stValve.xOPN_OK := iq_stValve.xEXT_OK AND iq_stValve.xAT_VAC;
END_IF

(* Valve operation *)
if NOT (iq_stValve.xOPN_OK) THEN iq_stValve.pv_xOPN_SW:= FALSE; END_IF // redundant??
(* Here's where the valve opens *)
iq_stValve.q_xOPN_DO := (iq_stValve.pv_xOPN_SW AND iq_stValve.xOPN_OK) OR (tonOvrd.Q AND i_xOverrideMode);
END_ACTION

ACTION ACT_ResetAlarms:
iq_stValve.xERR_DifPres R= iq_stValve.pv_xAlmRst;
iq_stValve.xERR_SP R= iq_stValve.pv_xAlmRst;
iq_stValve.bErrorPresent R= iq_stValve.pv_xAlmRst;

IF ( iq_stValve.pv_xAlmRst) THEN
	iq_stValve.sErrorMessage :='';
END_IF
END_ACTION

METHOD PUBLIC M_IsClosed : BOOL
VAR_INPUT
END_VAR
M_IsClosed := (This^.iq_stValve.eState = E_ValvePositionState.CLOSED);
END_METHOD

METHOD PUBLIC M_IsOpen : BOOL
VAR_INPUT
END_VAR
M_IsOpen := (This^.iq_stValve.eState = E_ValvePositionState.OPEN);
END_METHOD

// Use this Methode to Open or close the valve by setting the OPN_SW to the input value.
METHOD PUBLIC M_Set_OPN_SW : BOOL
VAR_INPUT
		value:BOOL;
END_VAR
This^.iq_stValve.pv_xOPN_SW := value;
END_METHOD

END_FUNCTION_BLOCK

// ---- POUs/FB_ValveBase.TcPOU
FUNCTION_BLOCK FB_ValveBase
VAR_INPUT
END_VAR
VAR_OUTPUT
END_VAR
VAR
	// For logging
    fbLogger : FB_LogMessage := (eSubsystem:=E_SubSystem.VACUUM);
   // ePrevState : E_ValvePositionState;
    tErrorPresent : R_TRIG;
    tAction : R_TRIG; // Primary action of this device (OPN_DO, etc.)
    tOverrideActivated : R_TRIG;
END_VAR

ACTION ACT_Logger:

END_ACTION

END_FUNCTION_BLOCK

// ---- POUs/FB_VRC_NO.TcPOU
(* This function block is different from the regular VRC in that CLOSING must be permitted. *)
FUNCTION_BLOCK FB_VRC_NO EXTENDS FB_ValveBase
VAR_IN_OUT

END_VAR
VAR_INPUT
	{attribute 'pytmc' := '
	pv: EXT_ILK_OK ;
	field: ZNAM NOT OK ;
	field: ONAM OK ;
	io: i ;
	'}
	i_xExtILK_OK : BOOL; //Connect to Interlock logic condition(e.g F_TURBO_VRC_ILK Function), otherwise, Set to True if the valve is not interlocked
	i_xOverrideMode : BOOL; (*To be linked to global override bit. This Overrides Vacuum logic only, EPS, MPS and PMPS are still enforces*)

END_VAR
VAR_OUTPUT
		iq_stValve : ST_VRC;
END_VAR
VAR

	{attribute 'noinit'}
	sPath: STRING;
	xFirstPass	:	BOOL;
	fbFSInit		:	R_TRIG;
	tonOvrd	:	TON;
	tonDelOK : TON;
	rtOK	:	R_TRIG;
	tOvrd	:	TIME := T#10s;
	(* Timeouts*)
	tTimeOutDuration: TIME:= T#10S;
	tOPNtimeout: TON;
	tCLStimeout:TON;
		{attribute 'pytmc' := '
	pv: CLS_SW ;
	field: ONAM CLOSE; 
	field: ZNAM OPEN;
	io: io ;
	'}
	pv_xCLS_SW	: BOOL;
	{attribute 'pytmc' := '
    pv: FORCE_CLS;
	io: io;
	'}
	pv_xOvrdCls	:	BOOL;

(*IO*)
	i_xOpnLS	AT%I*: BOOL;
	i_xClsLS	AT%I*: BOOL;
	q_xCLS_DO	AT%Q*: BOOL;

END_VAR

(* This function block is different from the regular VRC in that CLOSING must be permitted. *)

(* On first PLC pass, put valve into vented state, which implies a closed valve *)
fbFSInit( CLK := TRUE, Q => xFirstPass);
IF xFirstPass THEN
	pv_xCLS_SW := FALSE;
END_IF




///Check valve position
IF iq_stValve.i_xClsLS AND  iq_stValve.i_xOpnLS THEN
	iq_stValve.eState:=INVALID;
ELSIF NOT iq_stValve.i_xClsLS AND iq_stValve.i_xOpnLS AND iq_stValve.q_xOPN_DO THEN 
	iq_stValve.eState:=OPEN;
ELSIF iq_stValve.i_xClsLS AND NOT iq_stValve.i_xOpnLS AND NOT iq_stValve.q_xOPN_DO THEN 
	iq_stValve.eState:=CLOSED;
ELSIF NOT iq_stValve.i_xClsLS AND NOT iq_stValve.i_xOpnLS THEN 
	iq_stValve.eState:=MOVING;
ELSE
	iq_stValve.eState:=INVALID;
END_IF


(*evaluate Valve CLose external interlock*)
iq_stValve.xCLS_OK := i_xExtILK_OK;
IF NOT iq_stValve.xCLS_OK and NOT tonOvrd.Q THEN
	pv_xCLS_SW := FALSE;
END_IF


(* Override logic *)
(* Goal: give ability to override, but do so in a way that people won't forget it.
Solution: Override only after ten seconds of override, protect against blips,
when the valve permission goes true for more than ten seconds consistently, remove override
*)

tonDelOK(IN:=iq_stValve.xCLS_OK, PT:=T#10S);
rtOK(CLK:=tonDelOK.Q);
IF rtOK.Q AND pv_xOvrdCls THEN 
	pv_xOvrdCls :=FALSE; 
	if (iq_stValve.eState=CLOSED) AND (i_xOverrideMode) THEN pv_xCLS_SW := TRUE; END_IF
    //Log
    fbLogger(sMsg:='Override expired', eSevr:=TcEventSeverity.Warning);
END_IF

//Override timer
tonOvrd(IN:=pv_xOvrdCls, PT:=tOvrd);

(* Here's where the valve Actuates *)
q_xCLS_DO := ((iq_stValve.xCLS_OK  AND pv_xCLS_SW)OR (tonOvrd.Q AND i_xOverrideMode));
iq_stValve.q_xOPN_DO := NOT q_xCLS_DO;



///Check valve moving position timout
IF NOT iq_stValve.i_xClsLS AND tCLStimeout.Q THEN 
	iq_stValve.bErrorPresent := TRUE;
	//iq_stValve.sErrorMessage := ' Close Timeout';
ELSIF NOT iq_stValve.i_xOpnLS AND tOPNtimeout.Q THEN 
	iq_stValve.bErrorPresent := TRUE; 
	//iq_stValve.sErrorMessage := ' Open Timeout';
END_IF
IF (iq_stValve.eState=INVALID) THEN
	iq_stValve.bErrorPresent := TRUE; 
	//iq_stValve.sErrorMessage := CONCAT(sPath,' Invalid Valve Position');
END_IF

(*Timers*)
tOPNtimeout(IN:= iq_stValve.q_xOPN_DO, PT := tTimeOutDuration );
tCLStimeout(IN:= NOT iq_stValve.q_xOPN_DO, PT := tTimeOutDuration);


(*Soft IO Mapping*)
ACT_IO();

// Log States and triggers
ACT_Logger();

ACTION ACT_IO:
(*inputs*)
iq_stValve.i_xOpnLS := 	i_xOpnLS;
iq_stValve.i_xClsLS:=	i_xClsLS;
//iq_stValve. := i_xEXT_OK;
iq_stValve.xOverrideMode := i_xOverrideMode;
(*outputs*)
//q_xOPN_DO:= iq_stValve.q_xOPN_DO;
END_ACTION

METHOD PUBLIC M_IsClosed : BOOL
VAR_INPUT
END_VAR
M_IsClosed := (This^.iq_stValve.eState = E_ValvePositionState.CLOSED);
END_METHOD

METHOD PUBLIC M_IsOpen : BOOL
VAR_INPUT
END_VAR
M_IsOpen := (This^.iq_stValve.eState = E_ValvePositionState.OPEN);
END_METHOD

// Use this Methode to Open or close the valve by setting the OPN_SW to the input value.
METHOD PUBLIC M_Set_CLS_SW : BOOL
VAR_INPUT
		value:BOOL;
END_VAR
This^.pv_xCLS_SW := value;
END_METHOD

END_FUNCTION_BLOCK

// ---- POUs/FB_VGC_FFO.TcPOU
FUNCTION_BLOCK FB_VGC_FFO EXTENDS FB_VGC
VAR_INPUT
END_VAR
VAR_OUTPUT
	{attribute 'pytmc' := '
    pv: MPS_FAULT_OK
	field: ZNAM MPS FAULT ;
	field: ONAM MPS OK ;
	'}
	xMPS_OK:	BOOL; (*MPS Fast OK, is set when the Valve is Open*)

END_VAR
VAR_IN_OUT
	io_fbFFHWO    :    FB_HardwareFFOutput;
END_VAR
VAR
	// PMPS
	fbFF    :    FB_FastFault :=(
        i_DevName := 'VGC',
        i_Desc := 'Fault occurs when the valve is not in open state',
        i_TypeCode := 16#1010);
END_VAR



Super^.ACT_Init();
(*IO Mapping*)
Super^.ACT_IO();
Super^.A_Override();
Super^.A_PositionCheck();
Super^.A_Logger();
Super^.ACT_ResetAlarms();
Super^.A_EPS();
Super^.ACT_Main();
(*IO Mapping*)
Super^.ACT_IO();

(* When the valve  is open MPS is OK*)
xMPS_OK := (iq_stValve.eState=OPEN);//iq_stValve.i_xOpnLS; 
(*FAST FAULT*)
fbFF(i_xOK := xMPS_OK,
    i_xReset := i_xReset,
    io_fbFFHWO := io_fbFFHWO);

END_FUNCTION_BLOCK
